{attribute 'GeneratedUsingTerminal: EM3702-0000-0016'}
{attribute addProperty BoxType "EM3702-0000-0016"}
{attribute addProperty Id "EtcSlaveTerminalBaseAI_Input_Channel_1AT %I*AI_Input_Channel_5AF6604E8AI_Input_Channel_2AT %I*AI_Input_Channel_5AF6604E8WcStateAT %I*WcState_9091E0EB2InfoDataAT %I*InfoData_32EB74EA10"}
{attribute addProperty CRC "4246923465"}
{attribute addProperty Size "28"}
TYPE EM3702_FD22E8C9 EXTENDS EtcSlaveTerminalBase :
STRUCT
	{attribute addProperty Name "AI_Input_Channel_1"}
	AI_Input_Channel_1 : AI_Input_Channel_5AF6604E;
	{attribute addProperty Name "AI_Input_Channel_2"}
	AI_Input_Channel_2 : AI_Input_Channel_5AF6604E;
	{attribute addProperty Name "WcState"}
	WcState : WcState_9091E0EB;
	{attribute addProperty Name "InfoData"}
	InfoData : InfoData_32EB74EA;
END_STRUCT
END_TYPE

(* stored: Version 1.2.0.0, ProductVersion 3.1.4024.9
   DUT EM3702_FD22E8C9: Id {503bd23b-7845-4124-8b23-23ec61e0f020} *)
